// TwinCAT 3 PLC project SmartQualityControl_PLC
// ProgramVersion: 3.1.4024.12
// libraries:
//   Tc2_Standard, * (Beckhoff Automation GmbH)
//   Tc2_System, * (Beckhoff Automation GmbH)
//   Tc3_Module, * (Beckhoff Automation GmbH)
// project tree:
//   GVLs/ GVL_PythonBridge.TcGVL
//   / PlcTask.TcTTO
//   POUs/ MAIN.TcPOU
// real-time tasks:
//   TASK PlcTask: cycle T#10ms, priority 20, ADS port 350

CONFIGURATION SmartQualityControl_PLC
    RESOURCE PLC ON TwinCAT3
        TASK PlcTask(INTERVAL := T#10ms, PRIORITY := 20);
        PROGRAM MAIN WITH PlcTask : MAIN;
    END_RESOURCE
END_CONFIGURATION

// ---- GVLs/GVL_PythonBridge.TcGVL
VAR_GLOBAL
    // Python - PLC
    Start_Button        : BOOL;
    Emergency_Stop      : BOOL;
    Product_Sensor      : BOOL;
    Product_Defective   : BOOL;
    Stop_Line           : BOOL;
    Defect_Rate         : REAL;

    // PLC - Python
    Line_Running        : BOOL;
    Total_Count         : INT;
    Defect_Count        : INT;

    // Outputs
    Belt_Motor          : BOOL;
    Reject_Cylinder     : BOOL;
    Green_Light         : BOOL;
    Red_Light           : BOOL;
    Alarm_Buzzer        : BOOL;
END_VAR

// ---- POUs/MAIN.TcPOU
PROGRAM MAIN
VAR
    Timer_Inspection    : TON;
    Counter_Total       : CTU;
    Counter_Defect      : CTU;
    Product_Sensor_Rise : R_TRIG;
    Defect_Rise         : R_TRIG;
END_VAR

// --- Belt Motor Control ---
IF (GVL_PythonBridge.Start_Button OR GVL_PythonBridge.Belt_Motor)
   AND NOT GVL_PythonBridge.Emergency_Stop
   AND NOT GVL_PythonBridge.Stop_Line THEN
    GVL_PythonBridge.Belt_Motor   := TRUE;
    GVL_PythonBridge.Line_Running := TRUE;
ELSE
    GVL_PythonBridge.Belt_Motor   := FALSE;
    GVL_PythonBridge.Line_Running := FALSE;
END_IF;

// --- Inspection Timer ---
Timer_Inspection(IN := GVL_PythonBridge.Product_Sensor AND GVL_PythonBridge.Belt_Motor, PT := T#2S);

// --- Reject Cylinder ---
GVL_PythonBridge.Reject_Cylinder := Timer_Inspection.Q AND GVL_PythonBridge.Product_Defective;

// --- Indicator Lights ---
GVL_PythonBridge.Green_Light  := GVL_PythonBridge.Belt_Motor;
GVL_PythonBridge.Red_Light    := GVL_PythonBridge.Stop_Line;
GVL_PythonBridge.Alarm_Buzzer := GVL_PythonBridge.Stop_Line;

// --- Product Counter ---
Product_Sensor_Rise(CLK := GVL_PythonBridge.Product_Sensor);
Counter_Total.CU := Product_Sensor_Rise.Q;
Counter_Total.PV := 9999;
Counter_Total();
GVL_PythonBridge.Total_Count := Counter_Total.CV;

// --- Defect Counter ---
Defect_Rise(CLK := GVL_PythonBridge.Product_Defective);
Counter_Defect.CU := Defect_Rise.Q;
Counter_Defect.PV := 9999;
Counter_Defect();
GVL_PythonBridge.Defect_Count := Counter_Defect.CV;

// --- Auto Stop ---
IF GVL_PythonBridge.Defect_Rate >= 10.0 THEN
    GVL_PythonBridge.Stop_Line := TRUE;
END_IF;
IF GVL_PythonBridge.Start_Button AND GVL_PythonBridge.Stop_Line THEN
    GVL_PythonBridge.Stop_Line := FALSE;
END_IF;

END_PROGRAM
